FUNCTION_BLOCK FB_FT_INT (* Integrator *)
  (* Standard: OSCAT *)
  (* Version 0.0, 2011-07-27, 4DIAC-IDE, 4DIAC-Consortium *)
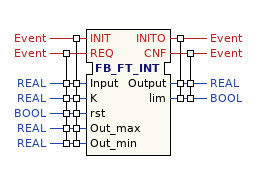
  EVENT_INPUT
    INIT WITH Input, K, rst, Out_max, Out_min; (* Initialization Request *)
    REQ WITH Input, K, rst, Out_max, Out_min; (* Normal Execution Request *)
  END_EVENT
  EVENT_OUTPUT
    INITO WITH Output, lim; (* Initialization Confirm *)
    CNF WITH Output, lim; (* Execution Confirmation *)
  END_EVENT
  VAR_INPUT
    Input : REAL; (* Input *)
    K : REAL; (* Amplification factor for Integrator *)
    rst : BOOL; (* Reset *)
    Out_max : REAL; (* Maximal output value *)
    Out_min : REAL; (* Minimal output value *)
  END_VAR
  VAR_OUTPUT
    Output : REAL; (* Output *)
    lim : BOOL; (* Returns true if the limit is exceeded *)
  END_VAR
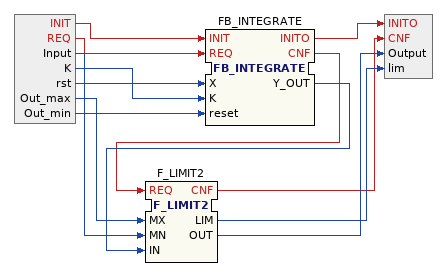
  FBS
    FB_INTEGRATE : FB_INTEGRATE;
    F_LIMIT2 : F_LIMIT2;
  END_FBS
  EVENT_CONNECTIONS
    INIT TO FB_INTEGRATE.INIT;
    REQ TO FB_INTEGRATE.REQ;
    FB_INTEGRATE.CNF TO F_LIMIT2.REQ;
    F_LIMIT2.CNF TO CNF;
    FB_INTEGRATE.INITO TO INITO;
  END_CONNECTIONS
  DATA_CONNECTIONS
    Input TO FB_INTEGRATE.X;
    K TO FB_INTEGRATE.K;
    rst TO FB_INTEGRATE.reset;
    Out_max TO F_LIMIT2.MX;
    Out_min TO F_LIMIT2.MN;
    FB_INTEGRATE.Y_OUT TO F_LIMIT2.IN;
    F_LIMIT2.LIM TO lim;
    F_LIMIT2.OUT TO Output;
  END_CONNECTIONS
END_FUNCTION_BLOCK
